FUNCTION_BLOCK ThreeConCtl (* Composite Function Block Type *)
  (* Standard: 61499-2 *)
  (* Version 0.2, 2003-12-05, JHC, Rockwell Automation, Renamed from NEWCOMPFB. *)
  (* Version 0.1, 2002-01-08, JHC, Rockwell Automation, Added DLY FB as example. *)
  (* Version 0.0, 2000-05-27, JHC, Rockwell Automation *)
  (* Compiler header: package fb.rt.conveyorIEC61499; *)
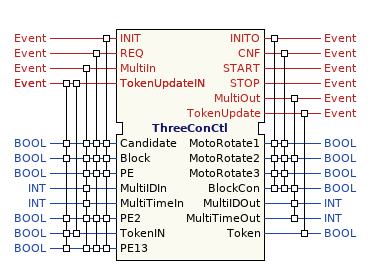
  EVENT_INPUT
    INIT WITH Candidate, Block, PE, PE2, PE13; (* Initialization Request *)
    REQ WITH Block, Candidate, PE, PE2, PE13; (* Normal Execution Request *)
    MultiIn WITH Candidate, Block, PE, MultiIDIn, MultiTimeIn, PE2, PE13;
    TokenUpdateIN WITH TokenIN;
    TokenUpdateIN WITH TokenIN, PE13, Candidate, Block, PE2;
  END_EVENT
  EVENT_OUTPUT
    INITO WITH MotoRotate1, MotoRotate2, MotoRotate3, BlockCon; (* Initialization Confirm *)
    CNF WITH MotoRotate1, MotoRotate2, MotoRotate3, BlockCon; (* Execution Confirmation *)
    START;
    STOP;
    MultiOut WITH MotoRotate2, BlockCon, MultiIDOut, MultiTimeOut;
    TokenUpdate WITH Token;
  END_EVENT
  VAR_INPUT
    Candidate : BOOL;
    Block : BOOL;
    PE : BOOL;
    MultiIDIn : INT;
    MultiTimeIn : INT;
    PE2 : BOOL;
    TokenIN : BOOL;
    PE13 : BOOL;
  END_VAR
  VAR_OUTPUT
    MotoRotate1 : BOOL;
    MotoRotate2 : BOOL;
    MotoRotate3 : BOOL;
    BlockCon : BOOL;
    MultiIDOut : INT;
    MultiTimeOut : INT;
    Token : BOOL;
  END_VAR
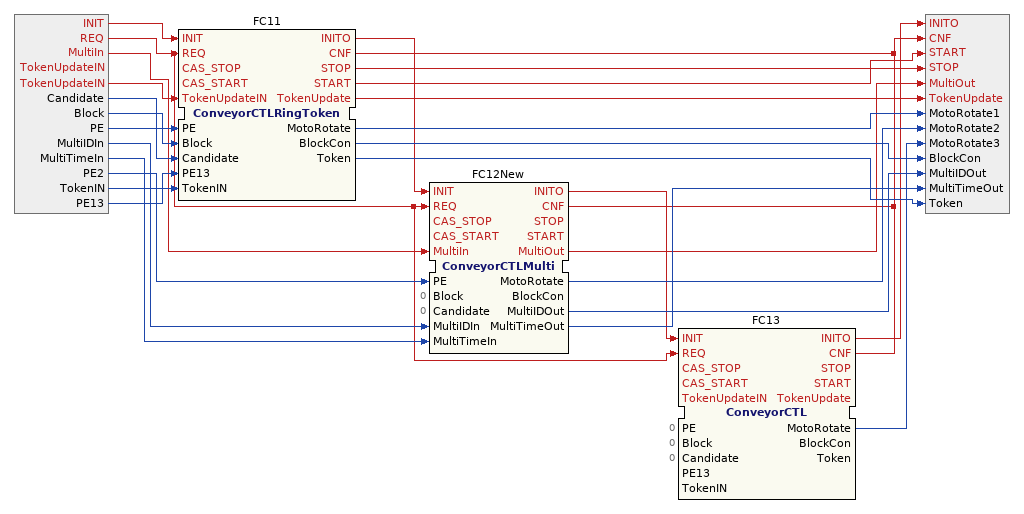
  FBS
    FC13 : ConveyorCTL(PE := 0, Block := 0, Candidate := 0);
    FC12New : ConveyorCTLMulti(Block := 0, Candidate := 0);
    FC11 : ConveyorCTLRingToken;
  END_FBS
  EVENT_CONNECTIONS
    FC13.INITO TO INITO;
    FC13.CNF TO CNF;
    REQ TO FC13.REQ;
    REQ TO FC12New.REQ;
    FC12New.CNF TO CNF;
    FC12New.INITO TO FC13.INIT;
    MultiIn TO FC12New.MultiIn;
    FC12New.MultiOut TO MultiOut;
    FC11.INITO TO FC12New.INIT;
    FC11.CNF TO CNF;
    FC11.STOP TO STOP;
    FC11.START TO START;
    INIT TO FC11.INIT;
    REQ TO FC11.REQ;
    FC11.TokenUpdate TO TokenUpdate;
    TokenUpdateIN TO FC11.TokenUpdateIN;
  END_CONNECTIONS
  DATA_CONNECTIONS
    FC13.MotoRotate TO MotoRotate3;
    FC12New.MotoRotate TO MotoRotate2;
    MultiIDIn TO FC12New.MultiIDIn;
    MultiTimeIn TO FC12New.MultiTimeIn;
    FC12New.MultiIDOut TO MultiIDOut;
    FC12New.MultiTimeOut TO MultiTimeOut;
    PE2 TO FC12New.PE;
    PE TO FC11.PE;
    Block TO FC11.Block;
    Candidate TO FC11.Candidate;
    FC11.MotoRotate TO MotoRotate1;
    FC11.BlockCon TO BlockCon;
    FC11.Token TO Token;
    PE13 TO FC11.PE13;
    TokenIN TO FC11.TokenIN;
  END_CONNECTIONS
END_FUNCTION_BLOCK
